Fanuc TP program (LS listing): CLOSE_T1.LS

/PROG  CLOSE_T1	  Macro
/ATTR
OWNER		= MNEDITOR;
COMMENT		= "";
PROG_SIZE	= 214;
CREATE		= DATE 25-07-07  TIME 18:41:28;
MODIFIED	= DATE 25-07-07  TIME 19:14:38;
FILE_NAME	= GRIPPER_;
VERSION		= 0;
LINE_COUNT	= 2;
MEMORY_SIZE	= 578;
PROTECT		= READ_WRITE;
TCD:  STACK_SIZE	= 0,
      TASK_PRIORITY	= 50,
      TIME_SLICE	= 0,
      BUSY_LAMP_OFF	= 0,
      ABORT_REQUEST	= 0,
      PAUSE_REQUEST	= 0;
DEFAULT_GROUP	= *,*,*,*,*;
CONTROL_CODE	= 00000000 00000000;
/APPL
/MN
   1:  RO[4:OFF:close T1]=ON ;
   2:  RO[3:ON :open T1]=OFF ;
/POS
/END
